// TwinCAT 3 PLC project PLC1_AssemblyLine
// Title: PLC1_AssemblyLine
// Company: Beckhoff Automation GmbH
// ProjectVersion: 1.0.0.0
// ProgramVersion: 3.1.4020.10
// libraries:
//   Tc2_MC2, * (Beckhoff Automation GmbH)
//   Tc2_Standard, * (Beckhoff Automation GmbH)
//   Tc2_System, * (Beckhoff Automation GmbH)
//   Tc3_EventLogger, * (Beckhoff Automation GmbH)
//   Tc3_Module, * (Beckhoff Automation GmbH)
// project tree:
//   DUTs/ E_FeederAutoState.TcDUT (not stored), E_AxisMode.TcDUT (not stored), E_StationState.TcDUT (not stored), ST_HmiAxisInfo.TcDUT (not stored), ST_HmiFeederInfo.TcDUT (not stored), ST_Hmi.TcDUT (not stored), ST_HmiAutomaticMode.TcDUT (not stored), ST_HmiErrorSimulation.TcDUT (not stored), ST_HmiFeederRecipe.TcDUT (not stored), ST_HmiManualMode.TcDUT (not stored), ST_HmiRecipeManagement.TcDUT (not stored), ST_PlcFeeder.TcDUT (not stored)
//   GVLs/ GVL.TcGVL (not stored)
//   / PlcTask.TcTTO (not stored)
//   POUs/ FB_Axis.TcPOU (not stored), FB_Feeder.TcPOU (not stored), MAIN.TcPOU
//   Version/ Global_Version.TcGVL (not stored)
// real-time tasks:
//   TASK PlcTask: cycle T#10ms, priority 8, ADS port 350
// motion (NC):
//   TASK NC-Task-SAF: cycle T#2ms, priority 4, ADS port 501
//   TASK NC-Task-SVB: cycle T#10ms, priority 10, ADS port 511
//   AXIS Feeder1_AxisX (id 1)
//     OtherSettings: AllowMotionCmdToSlave=true
//     encoder EncType=1
//       SoftEndMinControl: Enable=true
//       SoftEndMaxControl: Enable=true, Range=5000
//     drive DrvType=5
//       TimeComp: TaskDelayCycles=1
//     controller CtrType=1
//       CtrPara: PriorControlFactor=1
//         Observer: BandWidth=20
//   AXIS Feeder1_AxisY (id 2)
//     OtherSettings: AllowMotionCmdToSlave=true
//     encoder EncType=1
//       SoftEndMinControl: Enable=true
//       SoftEndMaxControl: Enable=true, Range=5000
//     drive DrvType=5
//       TimeComp: TaskDelayCycles=1
//     controller CtrType=1
//       CtrPara: PriorControlFactor=1
//         Observer: BandWidth=20
//   AXIS Feeder2_AxisX (id 3)
//     OtherSettings: AllowMotionCmdToSlave=true
//     encoder EncType=1
//       SoftEndMinControl: Enable=true
//       SoftEndMaxControl: Enable=true, Range=5000
//     drive DrvType=5
//       TimeComp: TaskDelayCycles=1
//     controller CtrType=1
//       CtrPara: PriorControlFactor=1
//         Observer: BandWidth=20
//   AXIS Feeder2_AxisY (id 4)
//     OtherSettings: AllowMotionCmdToSlave=true
//     encoder EncType=1
//       SoftEndMinControl: Enable=true
//       SoftEndMaxControl: Enable=true, Range=5000
//     drive DrvType=5
//       TimeComp: TaskDelayCycles=1
//     controller CtrType=1
//       CtrPara: PriorControlFactor=1
//         Observer: BandWidth=20
// variable links:
//   PLC1_AssemblyLine/PLC1_AssemblyLine Instance <-> NC-Task-SAF/Axes/Feeder1_AxisX
//     PlcTask Inputs/MAIN.fbFeeder1.stPlcFeeder.fbAxisX.stAxis.NcToPlc <-> Outputs/ToPlc
//     PlcTask Outputs/MAIN.fbFeeder1.stPlcFeeder.fbAxisX.stAxis.PlcToNc <-> Inputs/FromPlc
//   PLC1_AssemblyLine/PLC1_AssemblyLine Instance <-> NC-Task-SAF/Axes/Feeder1_AxisY
//     PlcTask Inputs/MAIN.fbFeeder1.stPlcFeeder.fbAxisY.stAxis.NcToPlc <-> Outputs/ToPlc
//     PlcTask Outputs/MAIN.fbFeeder1.stPlcFeeder.fbAxisY.stAxis.PlcToNc <-> Inputs/FromPlc
//   PLC1_AssemblyLine/PLC1_AssemblyLine Instance <-> NC-Task-SAF/Axes/Feeder2_AxisX
//     PlcTask Inputs/MAIN.fbFeeder2.stPlcFeeder.fbAxisX.stAxis.NcToPlc <-> Outputs/ToPlc
//     PlcTask Outputs/MAIN.fbFeeder2.stPlcFeeder.fbAxisX.stAxis.PlcToNc <-> Inputs/FromPlc
//   PLC1_AssemblyLine/PLC1_AssemblyLine Instance <-> NC-Task-SAF/Axes/Feeder2_AxisY
//     PlcTask Inputs/MAIN.fbFeeder2.stPlcFeeder.fbAxisY.stAxis.NcToPlc <-> Outputs/ToPlc
//     PlcTask Outputs/MAIN.fbFeeder2.stPlcFeeder.fbAxisY.stAxis.PlcToNc <-> Inputs/FromPlc

// ---- POUs/MAIN.TcPOU
PROGRAM MAIN
VAR
	fbFeeder1		: FB_Feeder(nFeederId := 1);
	fbFeeder2		: FB_Feeder(nFeederId := 2);
	bTest AT %I* : BOOL;
END_VAR

fbFeeder1();
fbFeeder2();

END_PROGRAM
